// TIA Portal V16 export
// export: Created 2024-09-05T17:40:15.417782Z, ExportSetting WithDefaults, DisplayName Totally Integrated Automation Portal, DisplayVersion V16 Update 6, DisplayName TIA Portal Version Control Interface, DisplayVersion V16 Update 2, DisplayName TIA Portal Openness, DisplayVersion V16 Update 6, DisplayName STEP 7 Professional, DisplayVersion V16 Update 6, DisplayName STEP 7 Safety, DisplayVersion V16, DisplayName WinCC Advanced, DisplayVersion V16 Update 6
TYPE "typeFbDiagnostics"
TITLE = typeDiagnosticsFBTemplate
// stored: IsFailsafeCompliant false
   STRUCT
      status : Word;   // Status of the FB or error identification when error occurred
      subfunctionStatus : DWord;   // Status or return value of called FBs, FCs and system blocks
   END_STRUCT;
END_TYPE
